(* IEC 61131-3 sources: crb-codesys/retrieval/output/codesys_repo/轴控/FB101_功能块/F06_收放卷应用, 8 files *)

(* ---- FB_卷径计算 copy 2.st ---- *)
FUNCTION_BLOCK FB_卷径计算
VAR_INPUT
   En  :BOOL;  (*使能功能块*)
   xMode :BOOL; (*FALSE*)
   xSet :BOOL;  (*初始化卷径*)
   Dir     :BOOL;   (*倒纸*)
   AxisDir :BOOL;  (*轴换向*)
   rDiaInit :REAL; (*初始卷径*)
   rDiaMax:REAL; (*最大卷径*)
   Length :REAL; (*采样长度*)
   rRatio :REAL; (*齿轮比，1.0*)
   MasterPos :LREAL; (*主轴当前位置*)
   SlavePos :LREAL;  (*从轴当前位置*)

END_VAR
VAR_OUTPUT
 RampDia:REAL;   (*斜坡后的可显示卷径*)
END_VAR
VAR
 fbR_TRIG: R_TRIG;
 rOldMasterPos:LREAL;
 rOldSlavePos:LREAL;
 rMasterLength:REAL;
 rSlaveLength:REAL;
 RAMP_REAL1: RAMP_REAL;
END_VAR
VAR_IN_OUT
 Diameter: REAL;  (*实时卷径*)
END_VAR

fbR_TRIG(CLK:=En , Q=> );
IF fbR_TRIG.Q THEN
    rOldMasterPos:=MasterPos;
    rOldSlavePos:=SlavePos;
END_IF

IF xSet THEN
    Diameter:=rDiaInit;
END_IF

IF NOT AxisDir AND NOT Dir AND En THEN
    IF SlavePos>rOldSlavePos+Length*rRatio THEN
        rMasterLength:=MasterPos-rOldMasterPos;
        rSlaveLength:=MasterPos-rOldSlavePos;
        Diameter:=rMasterLength/(3.14*rRatio);
        rOldMasterPos:=MasterPos;
        rOldSlavePos:=SlavePos;
    END_IF
END_IF
IF AxisDir AND NOT Dir AND En THEN
    IF SlavePos<rOldSlavePos-Length*rRatio THEN
        rMasterLength:=MasterPos-rOldMasterPos;
        rSlaveLength:=MasterPos-rOldSlavePos;
        Diameter:=rMasterLength/(3.14*rRatio);
        rOldMasterPos:=MasterPos;
        rOldSlavePos:=SlavePos;
    END_IF
END_IF

IF NOT AxisDir AND Dir AND En THEN
    IF SlavePos<rOldSlavePos-Length*rRatio THEN
        rMasterLength:=MasterPos-rOldMasterPos;
        rSlaveLength:=MasterPos-rOldSlavePos;
        Diameter:=rMasterLength/(3.14*rRatio);
        rOldMasterPos:=MasterPos;
        rOldSlavePos:=SlavePos;
    END_IF
END_IF
IF AxisDir AND Dir AND En THEN
    IF SlavePos>rOldSlavePos+Length*rRatio THEN
        rMasterLength:=MasterPos-rOldMasterPos;
        rSlaveLength:=MasterPos-rOldSlavePos;
        Diameter:=rMasterLength/(3.14*rRatio);
        rOldMasterPos:=MasterPos;
        rOldSlavePos:=SlavePos;
    END_IF
END_IF

RAMP_REAL1(
	IN:= ,
	ASCEND:= ,
	DESCEND:= ,
	TIMEBASE:= T#10MS,
	RESET:= ,
	OUT=> RampDia);

IF NOT xMode THEN
    RAMP_REAL1.ASCEND:=0.01;
    RAMP_REAL1.DESCEND:=0.005;
END_IF

IF xMode THEN
    RAMP_REAL1.ASCEND:=0.005;
    RAMP_REAL1.DESCEND:=0.01;
END_IF

IF xSet THEN
    RAMP_REAL1.ASCEND:=400;
    RAMP_REAL1.DESCEND:=400;
END_IF

(* ---- FB_卷径计算.st ---- *)
FUNCTION_BLOCK FB_卷径计算
VAR_INPUT
   En  :BOOL;  (*使能功能块*)
   xMode :BOOL; (*FALSE*)
   xSet :BOOL;  (*初始化卷径*)
   Dir     :BOOL;   (*倒纸*)
   AxisDir :BOOL;  (*轴换向*)
   rDiaInit :REAL; (*初始卷径*)
   rDiaMax:REAL; (*最大卷径*)
   Length :REAL; (*采样长度*)
   rRatio :REAL; (*齿轮比，1.0*)
   MasterPos :LREAL; (*主轴当前位置*)
   SlavePos :LREAL;  (*从轴当前位置*)

END_VAR
VAR_OUTPUT
 RampDia:REAL;   (*斜坡后的可显示卷径*)
END_VAR
VAR
 fbR_TRIG: R_TRIG;
 rOldMasterPos:LREAL;
 rOldSlavePos:LREAL;
 rMasterLength:REAL;
 rSlaveLength:REAL;
 RAMP_REAL1: RAMP_REAL;
END_VAR
VAR_IN_OUT
 Diameter: REAL;  (*实时卷径*)
END_VAR

fbR_TRIG(CLK:=En , Q=> );
IF fbR_TRIG.Q THEN
    rOldMasterPos:=MasterPos;
    rOldSlavePos:=SlavePos;
END_IF

IF xSet THEN
    Diameter:=rDiaInit;
END_IF

IF NOT AxisDir AND NOT Dir AND En THEN
    IF SlavePos>rOldSlavePos+Length*rRatio THEN
        rMasterLength:=MasterPos-rOldMasterPos;
        rSlaveLength:=MasterPos-rOldSlavePos;
        Diameter:=rMasterLength/(3.14*rRatio);
        rOldMasterPos:=MasterPos;
        rOldSlavePos:=SlavePos;
    END_IF
END_IF
IF AxisDir AND NOT Dir AND En THEN
    IF SlavePos<rOldSlavePos-Length*rRatio THEN
        rMasterLength:=MasterPos-rOldMasterPos;
        rSlaveLength:=MasterPos-rOldSlavePos;
        Diameter:=rMasterLength/(3.14*rRatio);
        rOldMasterPos:=MasterPos;
        rOldSlavePos:=SlavePos;
    END_IF
END_IF

IF NOT AxisDir AND Dir AND En THEN
    IF SlavePos<rOldSlavePos-Length*rRatio THEN
        rMasterLength:=MasterPos-rOldMasterPos;
        rSlaveLength:=MasterPos-rOldSlavePos;
        Diameter:=rMasterLength/(3.14*rRatio);
        rOldMasterPos:=MasterPos;
        rOldSlavePos:=SlavePos;
    END_IF
END_IF
IF AxisDir AND Dir AND En THEN
    IF SlavePos>rOldSlavePos+Length*rRatio THEN
        rMasterLength:=MasterPos-rOldMasterPos;
        rSlaveLength:=MasterPos-rOldSlavePos;
        Diameter:=rMasterLength/(3.14*rRatio);
        rOldMasterPos:=MasterPos;
        rOldSlavePos:=SlavePos;
    END_IF
END_IF

RAMP_REAL1(
	IN:= ,
	ASCEND:= ,
	DESCEND:= ,
	TIMEBASE:= T#10MS,
	RESET:= ,
	OUT=> RampDia);

IF NOT xMode THEN
    RAMP_REAL1.ASCEND:=0.01;
    RAMP_REAL1.DESCEND:=0.005;
END_IF

IF xMode THEN
    RAMP_REAL1.ASCEND:=0.005;
    RAMP_REAL1.DESCEND:=0.01;
END_IF

IF xSet THEN
    RAMP_REAL1.ASCEND:=400;
    RAMP_REAL1.DESCEND:=400;
END_IF

(* ---- FB_悬臂扭矩放卷.st ---- *)
FUNCTION_BLOCK FB_悬臂扭矩放卷
VAR_INPUT
END_VAR
VAR_OUTPUT
END_VAR
VAR
END_VAR

(* ---- FB_摆杆输出.st ---- *)
FUNCTION_BLOCK FB_摆杆输出
VAR_INPUT
	Enable:BOOL;
    摆臂的当前值:REAL;
    摆臂最小值:REAL;
    摆臂中间停止时最小值:REAL;
    摆臂中间停止时最大值:REAL;
    摆臂位置最大值:REAL;
    放卷的比例系数:REAL;
    收卷比例K值:REAL;
END_VAR
VAR_OUTPUT
	摆臂超过最大值报警:BOOL;
    放卷的输出值:REAL;
END_VAR
VAR
	正极片放卷值的变化:REAL;
    正极片临界值:DINT;
    摆臂收卷中间最大值:REAL;
    左边收卷区间:REAL;
    右边收卷区间:REAL;
END_VAR

IF Enable THEN
    摆臂收卷中间最大值:= (摆臂中间停止时最小值+摆臂最小值)/2;

    IF (摆臂的当前值<摆臂最小值) OR 摆臂的当前值<=0 THEN
         放卷的输出值:=0;(*停止输出*)

	      ELSIF (摆臂的当前值>=摆臂收卷中间最大值) AND (摆臂的当前值<摆臂中间停止时最小值) THEN
                  左边收卷区间:=摆臂中间停止时最小值-摆臂的当前值;
	              放卷的输出值:=左边收卷区间*收卷比例K值;  (*反转*)

          ELSIF (摆臂的当前值<摆臂收卷中间最大值) AND (摆臂的当前值>摆臂最小值) THEN
	              右边收卷区间:=摆臂的当前值-摆臂最小值;
	              放卷的输出值:=右边收卷区间*收卷比例K值;  (*反转*)

	      ELSIF (摆臂中间停止时最小值<=摆臂的当前值) AND (摆臂的当前值<摆臂中间停止时最大值) THEN
	              放卷的输出值:=0;  (*停止输出*)

          ELSIF (摆臂中间停止时最大值<=摆臂的当前值) AND (摆臂的当前值<摆臂位置最大值) THEN
		          放卷的输出值:=(放卷的比例系数*(摆臂的当前值-摆臂中间停止时最大值));  (*正转输出*int_to_real(正极片值-470)*正极片放卷值的变化*)

          ELSIF 摆臂位置最大值<=摆臂的当前值 THEN
			     摆臂超过最大值报警:=TRUE;

	END_IF;

END_IF;

(* ---- FB_线速度转角速度.st ---- *)
FUNCTION_BLOCK FB_线速度转角速度
VAR_INPUT
	Enble: BOOL;
	线速度: REAL; // m/min
	直径: REAL; // mm
	减速比: REAL;
END_VAR
VAR_OUTPUT
	角速度: REAL;
END_VAR
VAR
END_VAR

IF Enble THEN
	角速度:=1000.0*线速度*180.0/(60.0*3.14159265358979*((直径/1000.00)/2.0))*减速比;
END_IF;
// 1弧度=180°/π    弧角速度=V/R    角速度（°）=V/R*180°/π

(* ---- FB_角速度转线速度.st ---- *)
FUNCTION_BLOCK FB_角速度转线速度
VAR_INPUT
	Enble: BOOL;
	角速度: REAL;
	直径: REAL; // mm
	减速比: REAL;
END_VAR
VAR_OUTPUT
	线速度: REAL; // m/min
END_VAR
VAR
END_VAR

IF Enble THEN
	线速度:=LREAL_TO_REAL(角速度*(60.0*3.14159265358979*(直径/2.0))/(1000.0*180.0))/减速比;
END_IF;

(* ---- FB_速度同步.st ---- *)
FUNCTION_BLOCK FB_速度同步
VAR_INPUT
	Enble :BOOL;
    主轴速度 :REAL;
    主轴直径 :REAL;
    主轴减速比 :REAL;
    从轴直径 :REAL;
    从轴减速比 :REAL;
    速度系数 :REAL;
END_VAR
VAR_OUTPUT
	输出角速度: REAL;
END_VAR
VAR
END_VAR

IF Enble THEN
	输出角速度:=速度系数*主轴速度*(主轴直径*从轴减速比/(从轴直径*主轴减速比));
END_IF

(* ---- FB_锥度计算.st ---- *)
FUNCTION_BLOCK FB_锥度计算
VAR_INPUT
   rTensionSet   : REAL;       //张力设定
   rTaper        : REAL;       //锥度系数（1.0）
   rInit_Diameter  : REAL;    //最小卷径
   rAct_Diameter   : REAL;    //实时卷径
END_VAR
VAR_OUTPUT
   rTensionOut   : REAL;     //张力输出
END_VAR
VAR
END_VAR

rTensionOut:=rTensionSet*(1-rTaper*0.01*(1-rInit_Diameter/(rAct_Diameter+0.00001)));
